TYPE ST_EL3443_DPM_MUX_ULINT :
STRUCT
    nSelector : UINT := E_EL3443_DPM_Phase.Error_INDEX_Not_Valid;
    nValueRef : POINTER TO ULINT;
END_STRUCT
END_TYPE

(* stored: Version 1.1.0.1, ProductVersion 3.1.4024.12
   DUT ST_EL3443_DPM_MUX_ULINT: Id {5255343e-64f3-46e4-8391-a454ff8b7e8f} *)
